{attribute 'GeneratedUsingTerminal: EL3742-0000-0001'}
{attribute addProperty BoxType "EL3742-0000-0001"}
{attribute addProperty Id "EtcSlaveTerminalBaseCh1_CycleCountAT %I*Ch1_CycleCount_9DBE2BC52Ch1_Sample_0AT %I*Ch1_Sample_A71DD5012Ch2_CycleCountAT %I*Ch2_CycleCount_976A51B52Ch2_Sample_0AT %I*Ch2_Sample_9F6886E62WcStateAT %I*WcState_B516A2644InfoDataAT %I*InfoData_A7436BC610"}
{attribute addProperty CRC "155479622"}
{attribute addProperty Size "22"}
TYPE EL3742_09446E46 EXTENDS EtcSlaveTerminalBase :
STRUCT
	{attribute addProperty Name "Ch1_CycleCount"}
	Ch1_CycleCount : Ch1_CycleCount_9DBE2BC5;
	{attribute addProperty Name "Ch1_Sample_0"}
	Ch1_Sample_0 : Ch1_Sample_A71DD501;
	{attribute addProperty Name "Ch2_CycleCount"}
	Ch2_CycleCount : Ch2_CycleCount_976A51B5;
	{attribute addProperty Name "Ch2_Sample_0"}
	Ch2_Sample_0 : Ch2_Sample_9F6886E6;
	{attribute addProperty Name "WcState"}
	WcState : WcState_B516A264;
	{attribute addProperty Name "InfoData"}
	InfoData : InfoData_A7436BC6;
END_STRUCT
END_TYPE

(* stored: Version 1.2.0.0, ProductVersion 3.1.4024.9
   DUT EL3742_09446E46: Id {03570e41-81d3-4fa1-8372-9861223f2cd7} *)
